ABB RobotStudio station: Tp2_20201213-233457.rsstn

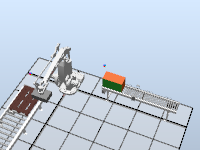
Station Tp2 (saved by RobotStudio 20.2.9116.0)
Controller Controlador1
  mechanical unit ROB_1: IRB660_180_315__01_2, 6 joints, base frame (0, 0, 0) mm
Layout (positions relative to the parent item):
  - transporteCajas [part, from Equipment\Conveyor Guide 400.rslib] at (0, 1500, 0) mm, rotated rx 0 ry 0 rz 90 deg
  - Euro Pallet [graphiccomponentgroup, from Equipment\Euro Pallet.rslib] at (1000, -1425, 435) mm
    - Body 1 [part, from Equipment\Euro Pallet.rslib]
  - transportePallets [part, from Equipment\Conveyor 950 4000 h2.rslib] at (1000, -1500, 0) mm
  - caja [part] at (-200, 1500, 770) mm
  - IRB660_180_315__01_2 [mechanism, from Robots\IRB660_180_315__01.rslib] at (0, 0, 0) mm; joint values [0, 0, 0, 0] (rad or m)
  - ventosa_tool [mechanism] at (1910, 0, 1833) mm, rotated rx 180 ry 0 rz 180 deg
      TCP ventosa_tool at (0, 0, 200) mm
      links: ventosa
  - basePallet [frame] at (1000, -1025, 435) mm
Attachment: Euro Pallet is attached to transportePallets
Attachment: basePallet is attached to Euro Pallet
Attachment: ventosa_tool is attached to IRB660_180_315__01_2 / Link6
EventTableEntry 2069: Group=, Trigger=do_pick 2070, Actions=[EventTableActionAttach 2071], Comment=, ActivationMode=2, Cyclic=false
EventTableTriggerIO 2070: IOValue=[1], IRC5Controller=? -1, Operator=0, SignalSource=Controlador1 1586
EventTableActionAttach 2071: AttachmentParent=ventosa_tool 1580, AttachmentChild=caja 1044, MountObject=false, Offset=[X=1, Y=0, Z=0, W=0, X=0, Y=1, Z=0, W=0, X=0, Y=0, Z=1, W=0, X=0, Y=0, Z=0, W=1], FlangeIndext=0, FindNearest=false
EventTableEntry 2072: Group=, Trigger=do_pick 2073, Actions=[EventTableActionDetach 2074], Comment=, ActivationMode=2, Cyclic=false
EventTableTriggerIO 2073: IOValue=[0], IRC5Controller=? -1, Operator=0, SignalSource=Controlador1 1586
EventTableActionDetach 2074: AttachmentParent=ventosa_tool 1580, AttachmentChild=caja 1044
Targets, tools, work objects and paths stored in the station, written as RAPID:
! task T_ROB1
MODULE Module1
  PERS tooldata ventosa_tool:=[TRUE,[[0,0,200],[1,0,0,0]],[1,[0,0,1],[1,0,0,0],0,0,0]];
  PERS wobjdata pistaCajas:=[FALSE,TRUE,"",[[-200,1500,770],[1,0,0,0]],[[0,0,0],[1,0,0,0]]];
  PERS wobjdata pistaPallets:=[FALSE,TRUE,"",[[1000,-1025,435],[1,0,0,0]],[[0,0,0],[1,0,0,0]]];
  CONST robtarget lugarEspera:=[[0,0,1000],[1,0,0,0],[0,0,0,0],[9E+09,9E+09,9E+09,9E+09,9E+09,9E+09]];
  CONST robtarget lugarEspera_2:=[[0,0,1000],[1,0,0,0],[0,0,0,0],[9E+09,9E+09,9E+09,9E+09,9E+09,9E+09]];
  PROC main()
  ENDPROC
  PROC esperarCaja()
  ENDPROC
ENDMODULE

